FUNCTION F_DetectOnlineChange : BOOL
VAR_STAT
    StoredOnlineChangeCnt : UDINT := 99;
END_VAR

F_DetectOnlineChange  := (TwinCAT_SystemInfoVarList._AppInfo.OnlineChangeCnt <> StoredOnlineChangeCnt);
StoredOnlineChangeCnt := TwinCAT_SystemInfoVarList._AppInfo.OnlineChangeCnt;

END_FUNCTION

(* stored: Version 1.1.0.1, ProductVersion 3.1.4024.12
   POU F_DetectOnlineChange: Id {4a5b4e3a-5eaa-41a7-8bb3-20de1a062cb9}, SpecialFunc None *)
